_CFC_ (* Continuous Function Chart, elements in execution order *)
(* 50с *)
#0 INT_TO_TIME(SHU6_P2_YA3_ZADER_RAS_DOST)
#1 MUL(#0, 1000)
#2 TON_YA3_Rassog1:TON(IN: YA3_DOST, PT: #1)
#3 ABS(SHU6_P2_YA3_RASSOG)
#4 GT(#3, SHU6_P2_YA3_UST_RASSOG)
#5 GT(SHU6_P2_YA3_RASSOG, SHU6_P2_YA3_UST_RASSOG)
#6 SEL(SHU6_P2_UST_RE_STOP, #4, #5)
#7 ABS(SHU6_P2_YA3_RASSOG_POL)
#8 GT(#7, SHU6_P2_YA3_UST_RASSOG)
#9 AND(TRUE, #8)
#10 YA3_REG_POL <= #9
#11 SEL(YA3_REG_POL, #6, #8)
#12 AND(NOT SHU6_P2_UST_RE_PUSK, #11)
#13 INT_TO_TIME(SHU6_P2_YA3_ZADER_RAS)
#14 MUL(#13, 1000)
#15 TON_YA3_Rassog:TON(IN: #12, PT: #14)
#16 OR(#15.Q, YA3_AO_OTKAZ)
#17 AND(#2.Q, SHU6_P2_YA3_SA4_DI1_A, #16)
#18 SR_YA3_Otk:SR(SET1: #17, RESET: SHU6_P2_SB)
#19 SHU6_P2_Z_YA3_OTKAZ <= #18.Q1
_END_CFC_
(* the same logic as Structured Text *)
(* 50с *)
TON_YA3_Rassog1(IN := YA3_DOST, PT := INT_TO_TIME(SHU6_P2_YA3_ZADER_RAS_DOST) * 1000);
_t14 := ABS(SHU6_P2_YA3_RASSOG_POL) > SHU6_P2_YA3_UST_RASSOG;
YA3_REG_POL := TRUE AND _t14;
TON_YA3_Rassog(IN := NOT SHU6_P2_UST_RE_PUSK AND SEL(YA3_REG_POL, SEL(SHU6_P2_UST_RE_STOP, ABS(SHU6_P2_YA3_RASSOG) > SHU6_P2_YA3_UST_RASSOG, SHU6_P2_YA3_RASSOG > SHU6_P2_YA3_UST_RASSOG), _t14), PT := INT_TO_TIME(SHU6_P2_YA3_ZADER_RAS) * 1000);
SR_YA3_Otk(SET1 := TON_YA3_Rassog1.Q AND SHU6_P2_YA3_SA4_DI1_A AND (TON_YA3_Rassog.Q OR YA3_AO_OTKAZ), RESET := SHU6_P2_SB);
SHU6_P2_Z_YA3_OTKAZ := SR_YA3_Otk.Q1;
END_PROGRAM

(* POU TZBiS/TZB/Z_YA4_Otk, CFC *)
PROGRAM Z_YA4_Otk
VAR
	RS_YA4_OTKZ: SR;

	UE3_ZADER: TON;
	SHU6_P2_YA4_AO1ER: TON;
	F_trig_ai: F_TRIG;
	TON_YA4: TON;
	YA4_ZADER_POL: TON;
	YA4_ZADER_TEMP: TON;
END_VAR
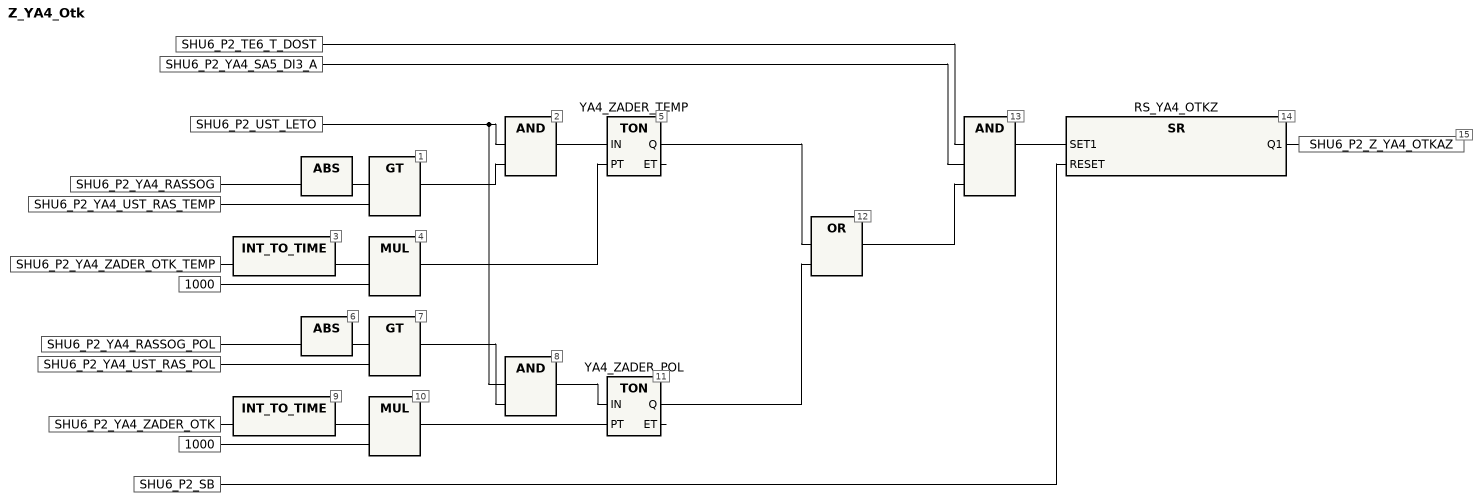
_CFC_ (* Continuous Function Chart, elements in execution order *)
#0 ABS(SHU6_P2_YA4_RASSOG)
#1 GT(#0, SHU6_P2_YA4_UST_RAS_TEMP)
#2 AND(SHU6_P2_UST_LETO, #1)
#3 INT_TO_TIME(SHU6_P2_YA4_ZADER_OTK_TEMP)
#4 MUL(#3, 1000)
#5 YA4_ZADER_TEMP:TON(IN: #2, PT: #4)
#6 ABS(SHU6_P2_YA4_RASSOG_POL)
#7 GT(#6, SHU6_P2_YA4_UST_RAS_POL)
#8 AND(SHU6_P2_UST_LETO, #7)
#9 INT_TO_TIME(SHU6_P2_YA4_ZADER_OTK)
#10 MUL(#9, 1000)
#11 YA4_ZADER_POL:TON(IN: #8, PT: #10)
#12 OR(#5.Q, #11.Q)
#13 AND(SHU6_P2_TE6_T_DOST, SHU6_P2_YA4_SA5_DI3_A, #12)
#14 RS_YA4_OTKZ:SR(SET1: #13, RESET: SHU6_P2_SB)
#15 SHU6_P2_Z_YA4_OTKAZ <= #14.Q1
_END_CFC_
(* the same logic as Structured Text *)
YA4_ZADER_TEMP(IN := SHU6_P2_UST_LETO AND (ABS(SHU6_P2_YA4_RASSOG) > SHU6_P2_YA4_UST_RAS_TEMP), PT := INT_TO_TIME(SHU6_P2_YA4_ZADER_OTK_TEMP) * 1000);
YA4_ZADER_POL(IN := SHU6_P2_UST_LETO AND (ABS(SHU6_P2_YA4_RASSOG_POL) > SHU6_P2_YA4_UST_RAS_POL), PT := INT_TO_TIME(SHU6_P2_YA4_ZADER_OTK) * 1000);
RS_YA4_OTKZ(SET1 := SHU6_P2_TE6_T_DOST AND SHU6_P2_YA4_SA5_DI3_A AND (YA4_ZADER_TEMP.Q OR YA4_ZADER_POL.Q), RESET := SHU6_P2_SB);
SHU6_P2_Z_YA4_OTKAZ := RS_YA4_OTKZ.Q1;
END_PROGRAM

(* POU TZBiS/TZB/Z_YA1_Otk, CFC *)
PROGRAM Z_YA1_Otk
VAR
	SR_YA2_Otkaz: SR;
	TON_YA2_Otk: TON;
	TON_YA2_N_OTKR: TON;
	TON_YA2_N_ZAKR: TON;
	TON_YA2_ZKR: TON;
	TON_AVT: TON;

	a: BOOL;
	b: BOOL;
	c: BOOL;
	d: BOOL;
	e: BOOL;
	TON_YA1_Otk: TON;
	TON_YA1_ZKR: TON;
	TON_YA1_N_OTKR: TON;
	TON_YA1_N_ZAKR: TON;
	SR_YA1_Otkaz: SR;
END_VAR
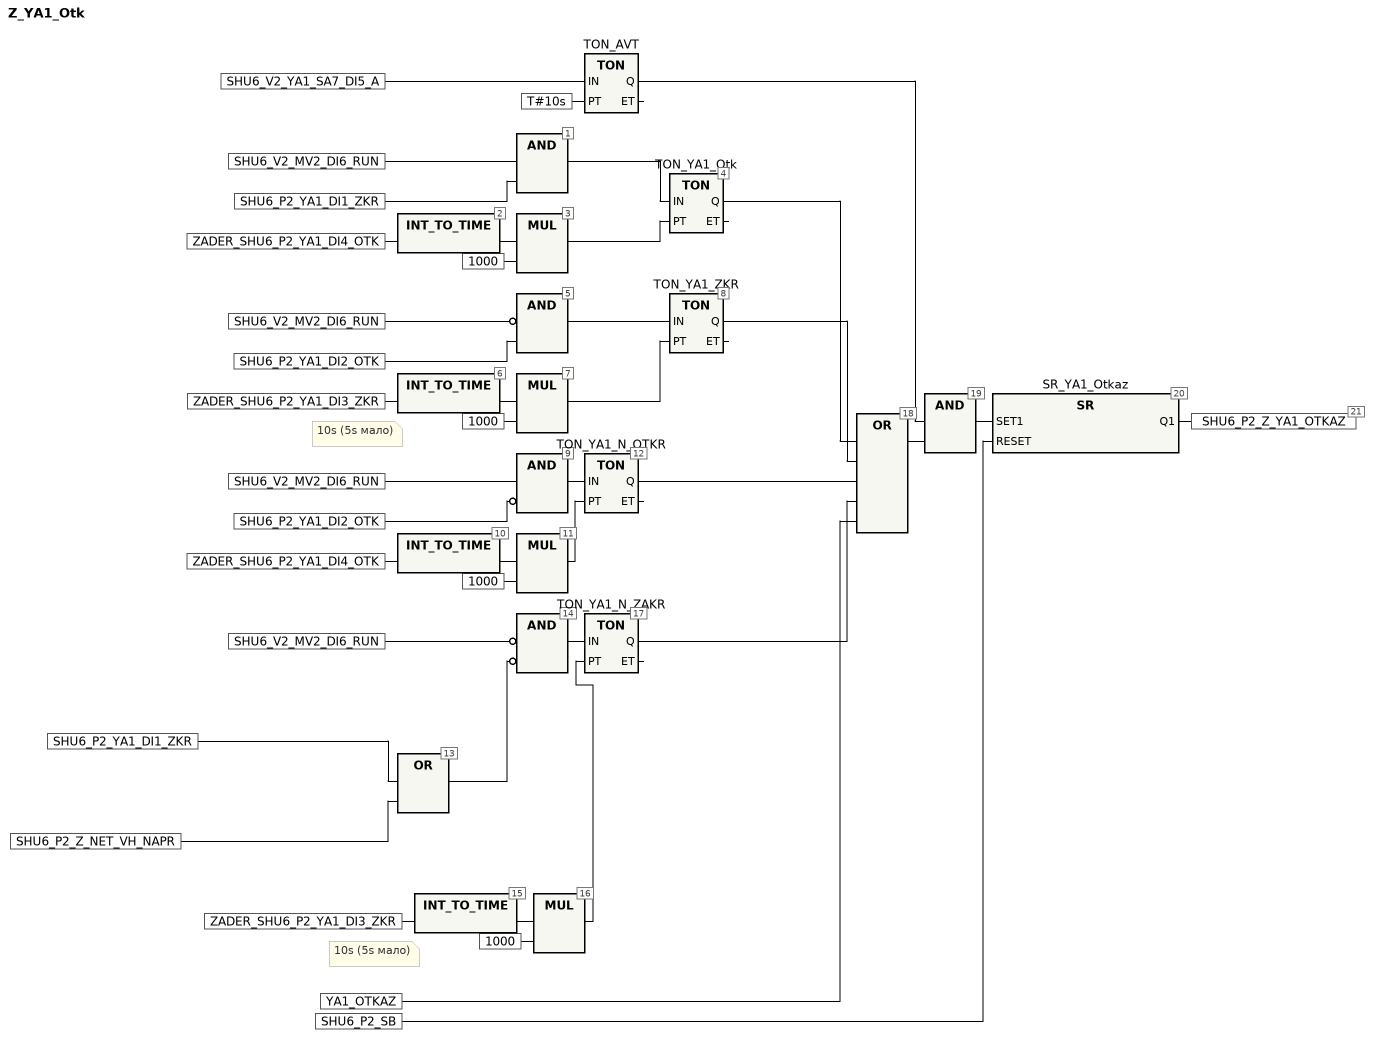
